FUNCTION_BLOCK ConveyorControl (* Decides Conveyor contorl *)
  (* Standard: 61499-2 *)
  (* Version 0.2, 2003-12-04, JHC, Rockwell Automation, Renamed for better indexing. *)
  (* Version 0.1, 2002-11-05, JHC, Rockwell Automation, Corrected missing ST element in Algorithm REQ. *)
  (* Version 0.0, 2000-05-30, JHC, Rockwell Automation *)
  (* Compiler header: package fb.rt.template; *)
  (* Compiler Java IBM Jikes 1.06 *)
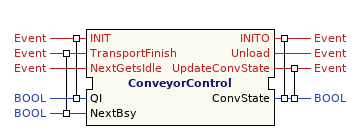
  EVENT_INPUT
    INIT WITH QI; (* Initialization Request *)
    TransportFinish WITH NextBsy; (* ConveyorEndsTransportationOfPallet *)
    NextGetsIdle;
  END_EVENT
  EVENT_OUTPUT
    INITO WITH ConvState; (* Initialization Confirm *)
    Unload;
    UpdateConvState WITH ConvState;
  END_EVENT
  VAR_INPUT
    QI : BOOL; (* Input event qualifier *)
    NextBsy : BOOL;
  END_VAR
  VAR_OUTPUT
    ConvState : BOOL; (* Output event qualifier *)
  END_VAR
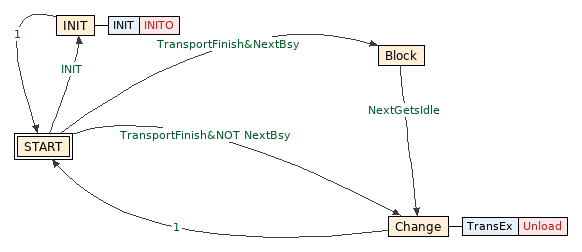
  EC_STATES
    START; (* Initial State *)
    INIT : INIT -> INITO; (* Initialization *)
    Change : TransEx -> Unload;
    Block;
  END_STATES
  EC_TRANSITIONS
    START TO INIT := INIT;
    INIT TO START := 1;
    Change TO START := 1;
    Block TO Change := NextGetsIdle;
    START TO Block := TransportFinish&NextBsy;
    START TO Change := TransportFinish&NOT NextBsy;
  END_TRANSITIONS
  ALGORITHM INIT IN ST: (* Initialization algorithm *)

  END_ALGORITHM
  ALGORITHM TransEx IN ST: (* Normally executed algorithm *)
ConvState := TRUE;
  END_ALGORITHM
END_FUNCTION_BLOCK
